// TIA Portal V16 export
// export: Created 2022-01-20T18:36:28.4625315Z, ExportSetting WithDefaults, DisplayName Totally Integrated Automation Portal, DisplayVersion V16, DisplayName TIA Portal Version Control Interface, DisplayVersion V16, DisplayName TIA Portal Openness, DisplayVersion V16, DisplayName STEP 7 Professional, DisplayVersion V16, DisplayName STEP 7 Safety, DisplayVersion V16, DisplayName WinCC Advanced, DisplayVersion V16
DATA_BLOCK "DB_Connect"   // DB2
{ S7_Optimized_Access := 'TRUE' }
// stored: AutoNumber true, InstanceOfName TCON_IP_v4, OfSystemLibElement TCON_IP_v4, OfSystemLibVersion 1.0
"TCON_IP_v4"
   // VAR
   //    InterfaceId : HW_ANY := 64;
   //    ID : CONN_OUC := 1;
   //    ConnectionType : Byte;
   //    ActiveEstablished : Bool := false;
   //    RemoteAddress { S7_SetPoint := 'True'} : IP_V4;
   //    RemotePort : UInt := 0;
   //    LocalPort : UInt := 5000;
   // END_VAR
BEGIN
   RemoteAddress.ADDR[1] := 192;
   RemoteAddress.ADDR[2] := 168;
   RemoteAddress.ADDR[3] := 1;
   RemoteAddress.ADDR[4] := 43;
END_DATA_BLOCK
